ABB RAPID module: Wobj_wobj_A2.mod

MODULE Wobj_wobj_A2
	! Points are read in order of declaration.
  ! Please do not change the order of points!

  LOCAL PERS robtarget pWobj_U_PointX1:=[[1214.12,-2047.981,-595.6802],[0.00630221795290709,-0.720875442028046,0.693015277385712,-0.00535879516974092],[-1,0,2,0],[0,9E+09,9E+09,9E+09,9E+09,9E+09]];
	LOCAL PERS robtarget pWobj_U_PointX2:=[[1796.117,-2027.769,-595.697],[0.00630304869264364,-0.720876812934875,0.693013906478882,-0.0053527201525867],[-1,0,2,0],[0,9E+09,9E+09,9E+09,9E+09,9E+09]];
	LOCAL PERS robtarget pWobj_U_PointY1:=[[1185.326,-1417.662,-595.6747],[0.00630108080804348,-0.72088223695755,0.693008184432983,-0.00536185363307595],[-1,0,2,0],[0,9E+09,9E+09,9E+09,9E+09,9E+09]];

ENDMODULE
